TYPE ST125_Recipe_t :
STRUCT
    xUseVerLeft           : BOOL; // Is the left vertical picker element is used
    xUseVerRight          : BOOL; // Is the right vertical picker element is used
    FeederConfig          : FeederDelays_t;
    diPieceGoodMaxHeight  : DINT; // Good piece maximum value (value is the output of the analog board)
    diPieceGoodMinHeight  : DINT; // Good piece minimum value (value is the output of the analog board)
    diPieceWrongMaxHeight : DINT; // Bad piece maximum value (value is the output of the analog board)
    diPieceWrongMinHeight : DINT; // Bad piece minimum value (value is the output of the analog board)
    TON_WaitPieceTime     : DINT; // additionnal waiting time of a piece to ensure the mesure is done correctly
    kraft_left_raw        : REAL; // force limit for left pnp, raw value
    kraft_right_raw       : REAL; // force limit for right pnp, raw value
END_STRUCT
END_TYPE

(* stored: Version 1.1.0.1, ProductVersion 3.1.4024.6
   DUT ST125_Recipe_t: Id {01370c0a-eb7d-4b76-9605-310d55798193} *)
